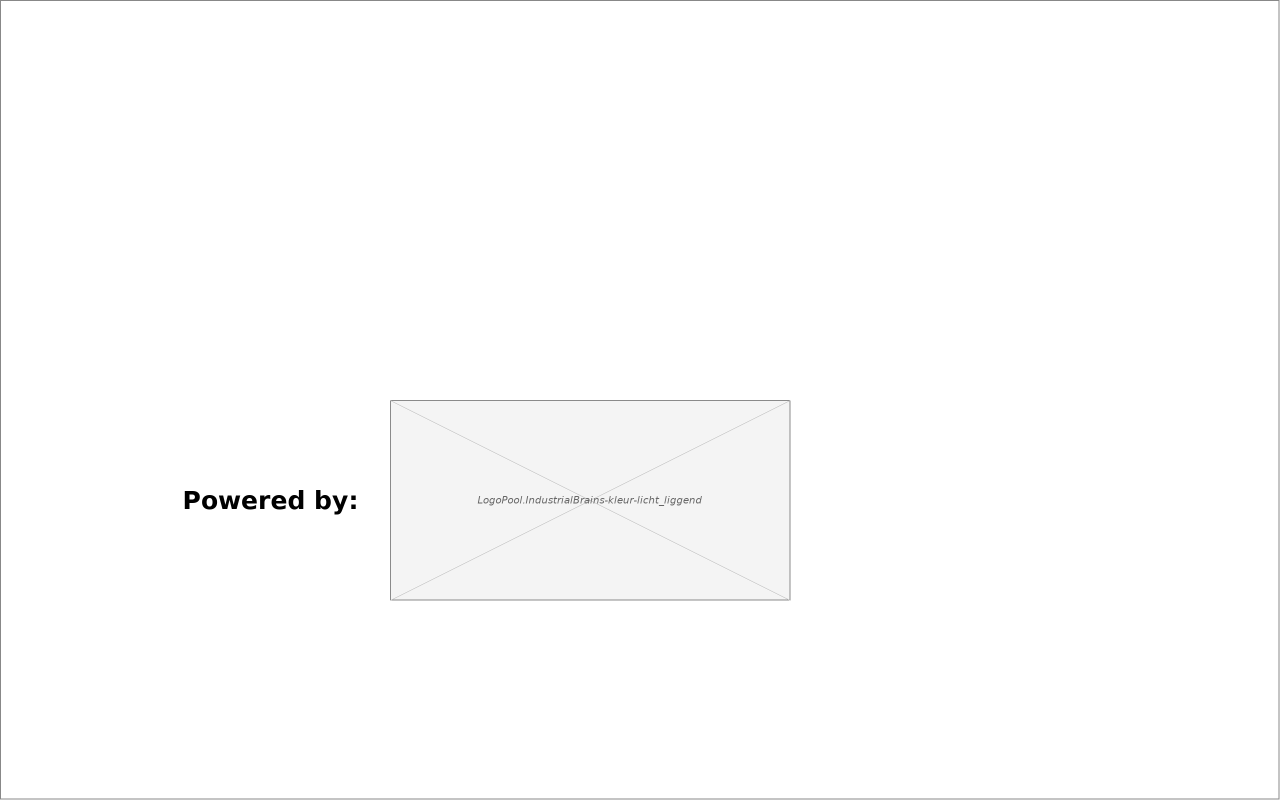
VISUALIZATION BackgroundLogoIB  // 1280x800
    Image (390,400 400x200), image: LogoPool.IndustrialBrains-kleur-licht_liggend
    Label (170,400 200x200), "Powered by:"
END_VISUALIZATION

(* stored: Version 1.1.0.1, ProductVersion 3.1.4024.11
   Visu BackgroundLogoIB: Id {f427881c-2361-4f1e-af47-55639561266d} *)
